FUNCTION_BLOCK AUDI_FB_CTUD (* Up-Down counter (UDINT) AUDI-Adapter Version *)
  (* Standard: 61499-2; Description: Copyright (c) 2026 Meisterschulen am Ostbahnhof This program and the accompanying materials are made available under the terms of the Eclipse Public License 2.0 which is available at https://www.eclipse.org/legal/epl-2.0/ SPDX-License-Identifier: EPL-2.0 NOTE: This block fires the AX output events (QU.E1, QD.E1) on every update (CU, CD, R, LD, PV). If on-change triggering is required, use of an AX_D_FF as a filter is recommended. *)
  (* Version 1.0, 2026-04-21, Franz Höpfinger, Meisterschulen am Ostbahnhof, initial API and implementation and/or initial documentation *)
  PACKAGE adapter::iec61131::counters;
  IMPORT eclipse4diac::core::TypeHash;
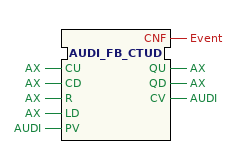
  EVENT_OUTPUT
    CNF; (* Execution Confirmation *)
  END_EVENT
  SOCKETS
    CU : adapter::types::unidirectional::AX; (* Count up *)
    CD : adapter::types::unidirectional::AX; (* Count down *)
    R : adapter::types::unidirectional::AX; (* Reset *)
    LD : adapter::types::unidirectional::AX; (* Load *)
    PV : adapter::types::unidirectional::AUDI; (* Preset value *)
  END_SOCKETS
  PLUGS
    QU : adapter::types::unidirectional::AX; (* Output Up *)
    QD : adapter::types::unidirectional::AX; (* Output Down *)
    CV : adapter::types::unidirectional::AUDI; (* Count value *)
  END_PLUGS
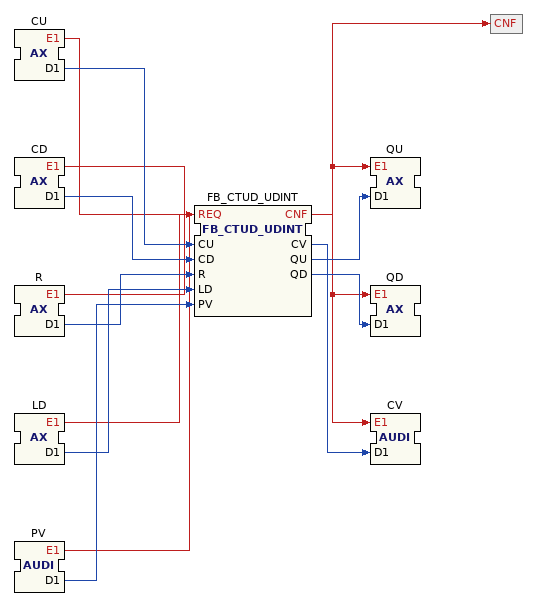
  FBS
    FB_CTUD_UDINT : iec61131::counters::FB_CTUD_UDINT;
  END_FBS
  EVENT_CONNECTIONS
    CU.E1 TO FB_CTUD_UDINT.REQ;
    CD.E1 TO FB_CTUD_UDINT.REQ;
    R.E1 TO FB_CTUD_UDINT.REQ;
    LD.E1 TO FB_CTUD_UDINT.REQ;
    PV.E1 TO FB_CTUD_UDINT.REQ;
    FB_CTUD_UDINT.CNF TO CV.E1;
    FB_CTUD_UDINT.CNF TO QU.E1;
    FB_CTUD_UDINT.CNF TO QD.E1;
    FB_CTUD_UDINT.CNF TO CNF;
  END_CONNECTIONS
  DATA_CONNECTIONS
    CU.D1 TO FB_CTUD_UDINT.CU;
    CD.D1 TO FB_CTUD_UDINT.CD;
    R.D1 TO FB_CTUD_UDINT.R;
    LD.D1 TO FB_CTUD_UDINT.LD;
    PV.D1 TO FB_CTUD_UDINT.PV;
    FB_CTUD_UDINT.CV TO CV.D1;
    FB_CTUD_UDINT.QU TO QU.D1;
    FB_CTUD_UDINT.QD TO QD.D1;
  END_CONNECTIONS
END_FUNCTION_BLOCK
